FUNCTION_BLOCK FB_CFC_SamplePOU
VAR_INPUT
//	eOperation	: INT;
	eOperation	: E_Operation;
END_VAR
VAR_OUTPUT
	iResultC	: DINT;
END_VAR
VAR
	arrDataA	: ARRAY [1..iMax] OF DINT;
	arrDataB	: ARRAY [1..iMax] OF DINT;
	arrDataC	: ARRAY [1..iMax] OF DINT;
	I 			: DINT;
	bInit		: BOOL := TRUE;
END_VAR
VAR CONSTANT
	iMax 		: DINT := 10;
END_VAR
VAR // added by the converter: edge detectors and wires of the graphical bodies
    _w1, _w2, _w4, _w6, _w9 : DINT;
    _w3, _w5, _w8 : ANY;
    _w7 : BOOL;
END_VAR

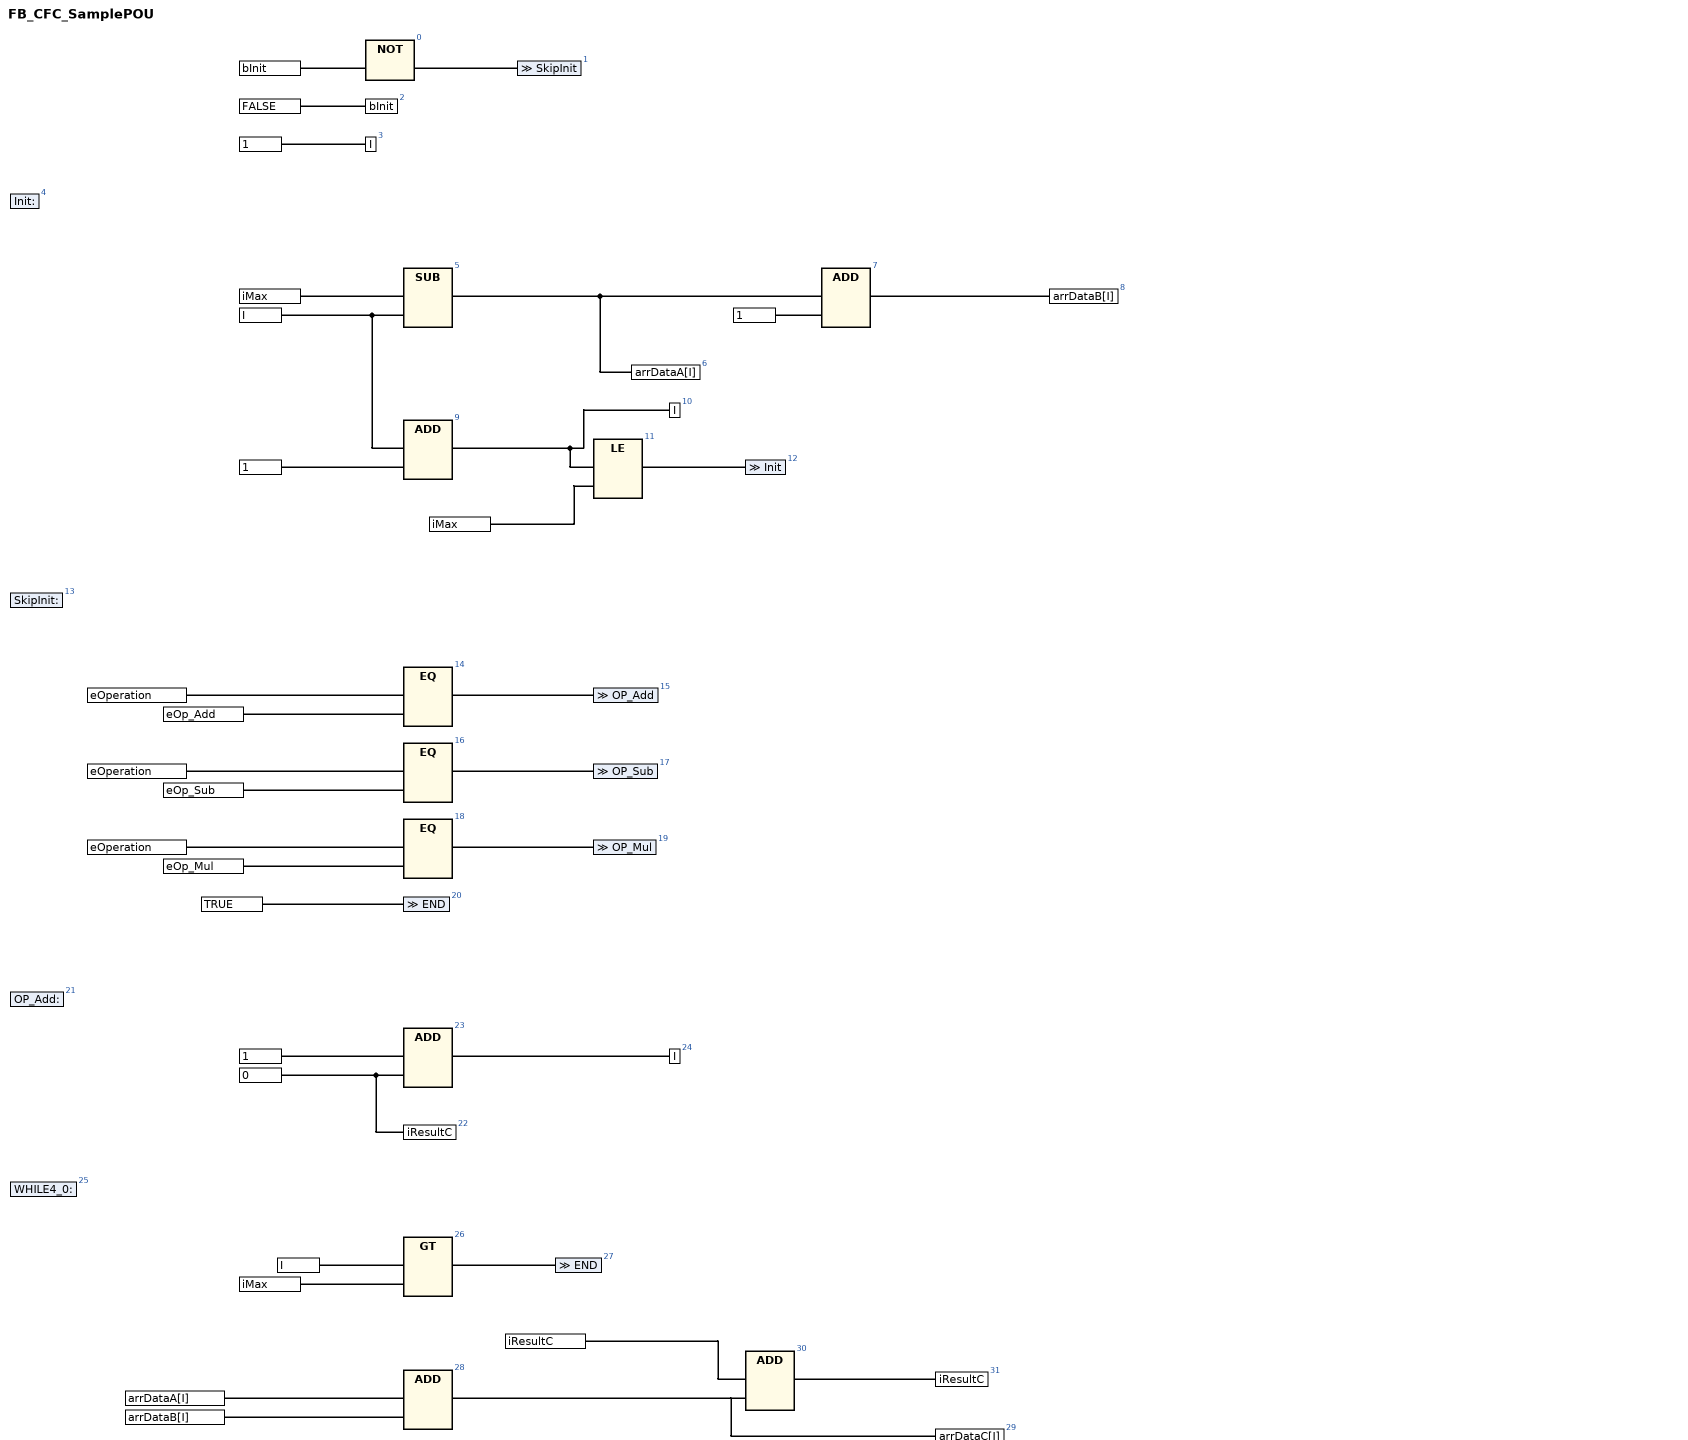
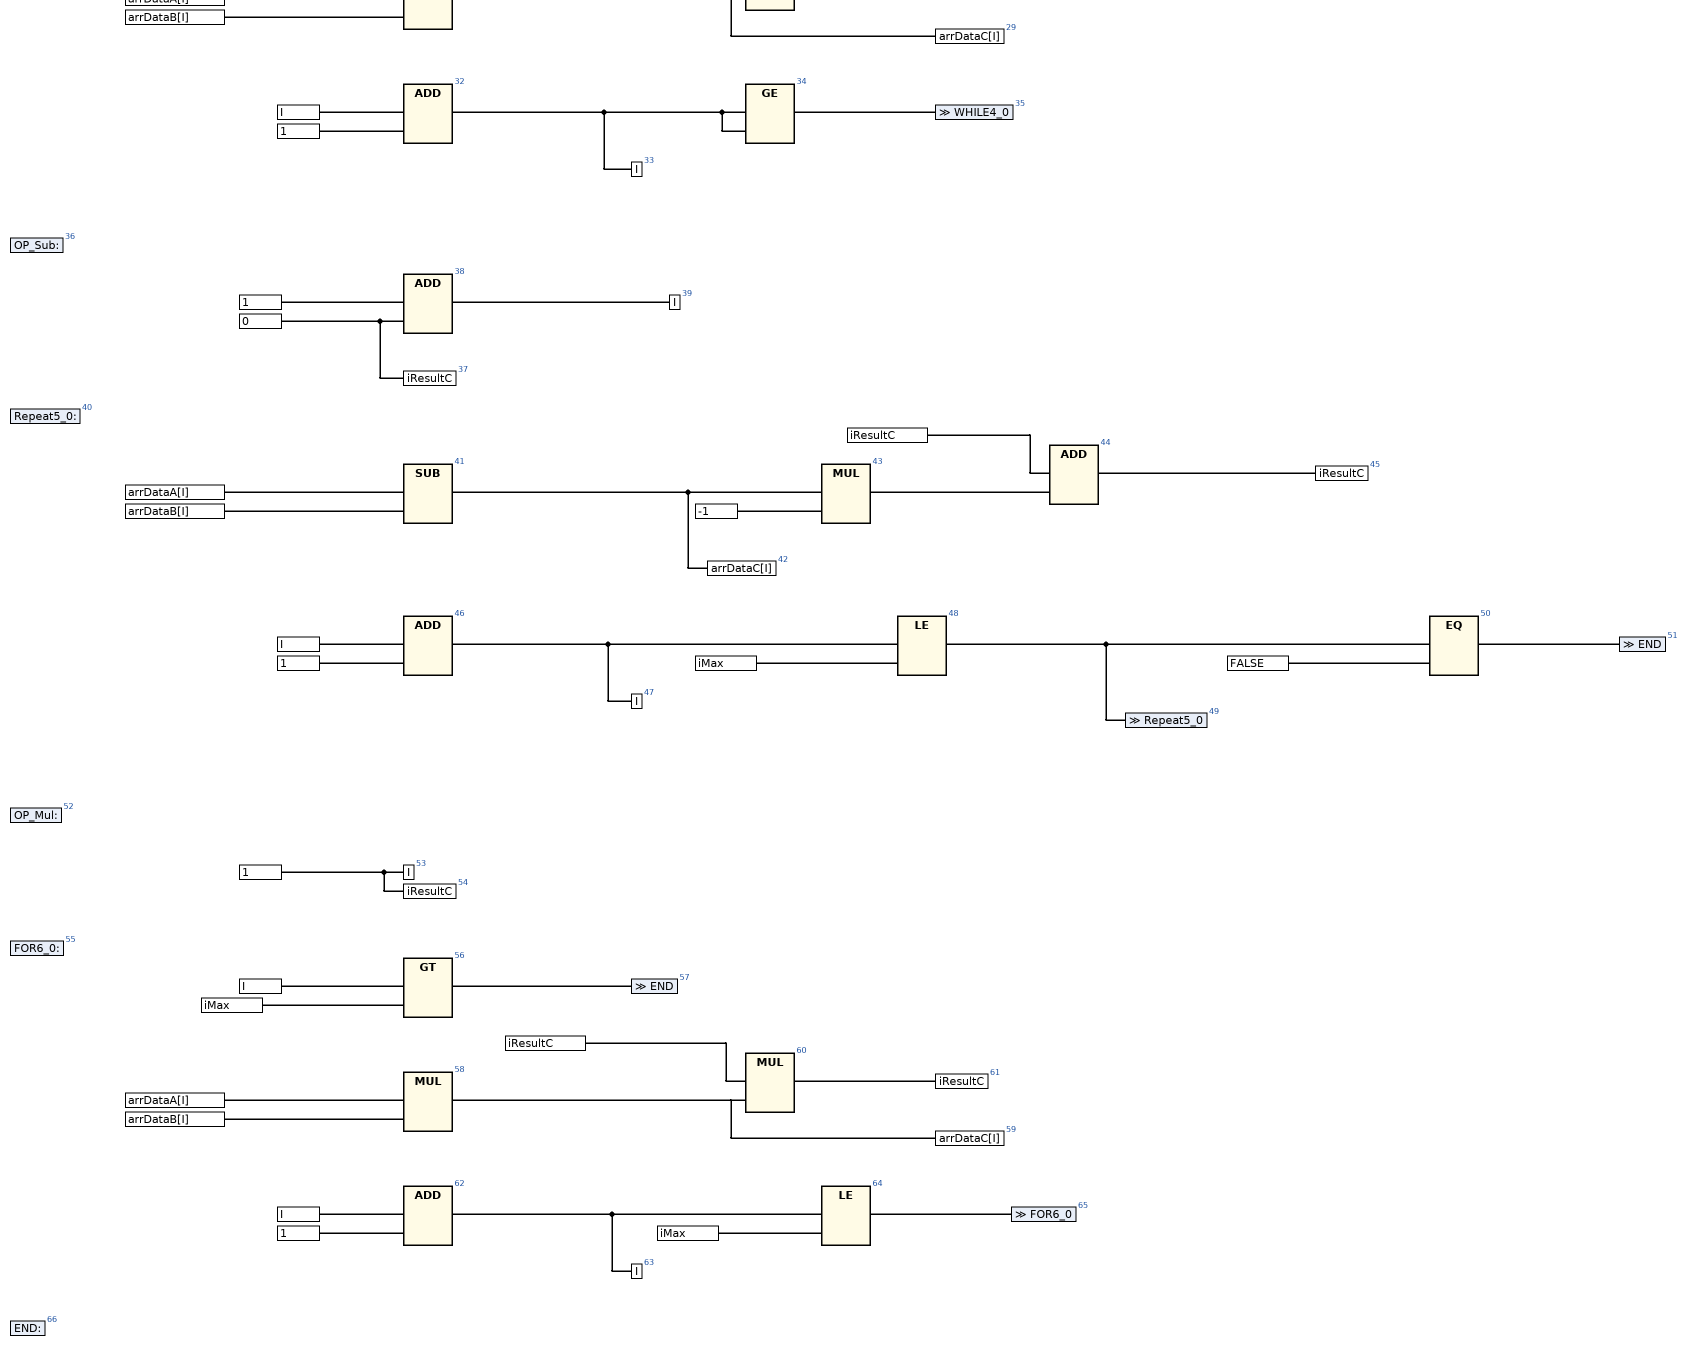
IF NOT bInit THEN JMP SkipInit; END_IF
bInit := FALSE;
I := 1;
Init: ;
_w1 := iMax - I;
arrDataA[I] := _w1;
arrDataB[I] := _w1 + 1;
_w2 := I + 1;
I := _w2;
IF _w2 <= iMax THEN JMP Init; END_IF
SkipInit: ;
IF eOperation = eOp_Add THEN JMP OP_Add; END_IF
IF eOperation = eOp_Sub THEN JMP OP_Sub; END_IF
IF eOperation = eOp_Mul THEN JMP OP_Mul; END_IF
IF TRUE THEN JMP END; END_IF
OP_Add: ;
iResultC := 0;
I := 1 + 0;
WHILE4_0: ;
IF I > iMax THEN JMP END; END_IF
_w3 := arrDataA[I] + arrDataB[I];
arrDataC[I] := _w3;
iResultC := iResultC + _w3;
_w4 := I + 1;
I := _w4;
IF _w4 >= _w4 THEN JMP WHILE4_0; END_IF
OP_Sub: ;
iResultC := 0;
I := 1 + 0;
Repeat5_0: ;
_w5 := arrDataA[I] - arrDataB[I];
arrDataC[I] := _w5;
iResultC := iResultC + _w5 * -1;
_w6 := I + 1;
I := _w6;
_w7 := _w6 <= iMax;
IF _w7 THEN JMP Repeat5_0; END_IF
IF _w7 = FALSE THEN JMP END; END_IF
OP_Mul: ;
I := 1;
iResultC := 1;
FOR6_0: ;
IF I > iMax THEN JMP END; END_IF
_w8 := arrDataA[I] * arrDataB[I];
arrDataC[I] := _w8;
iResultC := iResultC * _w8;
_w9 := I + 1;
I := _w9;
IF _w9 <= iMax THEN JMP FOR6_0; END_IF
END: ;

END_FUNCTION_BLOCK

(* stored: Version 1.1.0.1, ProductVersion 3.1.4024.11
   POU FB_CFC_SamplePOU: Id {7351355f-6984-4ef3-8ea0-8c200a229ead}, SpecialFunc None *)
